SUBAPPLICATION Uebung_221 (* Standard IEC 61131-3 FB_CTUD_DINT (Vor-/Rückwärtszähler, DINT) mit Terminal-Ausgabe *)
  (* Standard: 61131-3; Description: Copyright (c) 2026 Meisterschulen am Ostbahnhof This program and the accompanying materials are made available under the terms of the Eclipse Public License 2.0 which is available at https://www.eclipse.org/legal/epl-2.0/ SPDX-License-Identifier: EPL-2.0 *)
  (* Version 1.1, 2026-04-21, Franz Höpfinger, Meisterschulen am Ostbahnhof, Added terminal output for counter value *)
  (* Version 1.0, 2026-04-20, Franz Höpfinger, Meisterschulen am Ostbahnhof, initial API and implementation (IEC 61131-3 version) *)
  PACKAGE Uebungen;
  IMPORT Uebungen::const::UT::DefaultPool::OutputNumber_N1;
  IMPORT logiBUS::io::DI::logiBUS_DI::Input_I1;
  IMPORT logiBUS::io::DI::logiBUS_DI::Input_I2;
  IMPORT logiBUS::io::DI::logiBUS_DI::Input_I3;
  IMPORT logiBUS::io::DI::logiBUS_DI::Input_I4;
  IMPORT logiBUS::io::DQ::logiBUS_DO::Output_Q1;
  IMPORT logiBUS::io::DQ::logiBUS_DO::Output_Q2;
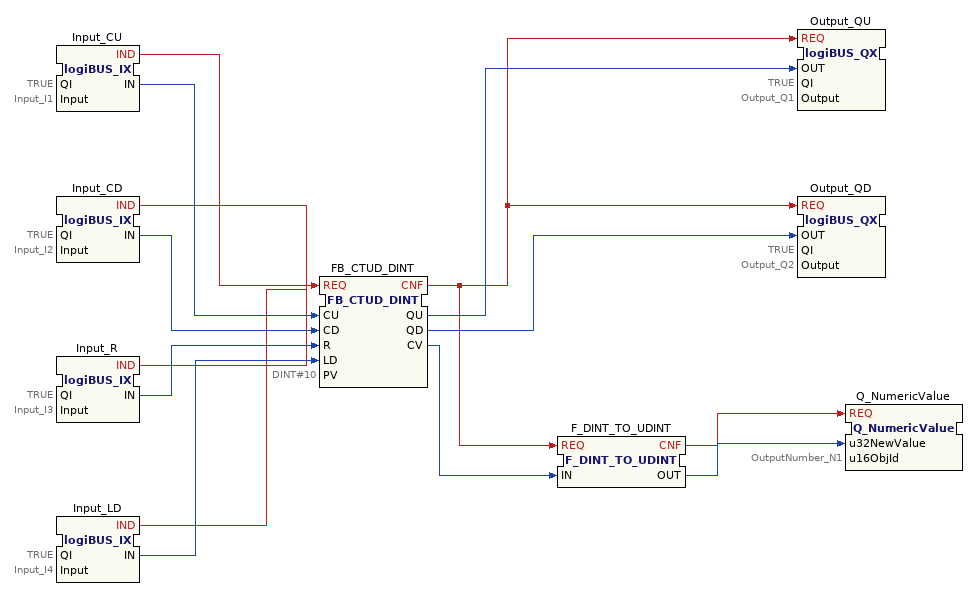
  (* F_DINT_TO_UDINT ist großer Quatsch ... keine Negativen Zahlen möglich *)
  FBS
    FB_CTUD_DINT : iec61131::counters::FB_CTUD_DINT(PV := DINT#10);
    Input_CU : logiBUS::io::DI::logiBUS_IX(QI := TRUE, Input := Input_I1);
    Input_CD : logiBUS::io::DI::logiBUS_IX(QI := TRUE, Input := Input_I2);
    Input_R : logiBUS::io::DI::logiBUS_IX(QI := TRUE, Input := Input_I3);
    Input_LD : logiBUS::io::DI::logiBUS_IX(QI := TRUE, Input := Input_I4);
    Output_QU : logiBUS::io::DQ::logiBUS_QX(QI := TRUE, Output := Output_Q1);
    Output_QD : logiBUS::io::DQ::logiBUS_QX(QI := TRUE, Output := Output_Q2);
    Q_NumericValue : isobus::UT::Q::Q_NumericValue(u16ObjId := OutputNumber_N1);
    F_DINT_TO_UDINT : iec61131::conversion::F_DINT_TO_UDINT;
  END_FBS
  EVENT_CONNECTIONS
    Input_CU.IND TO FB_CTUD_DINT.REQ;
    Input_CD.IND TO FB_CTUD_DINT.REQ;
    Input_R.IND TO FB_CTUD_DINT.REQ;
    Input_LD.IND TO FB_CTUD_DINT.REQ;
    FB_CTUD_DINT.CNF TO Output_QU.REQ;
    FB_CTUD_DINT.CNF TO Output_QD.REQ;
    FB_CTUD_DINT.CNF TO F_DINT_TO_UDINT.REQ;
    F_DINT_TO_UDINT.CNF TO Q_NumericValue.REQ;
  END_CONNECTIONS
  DATA_CONNECTIONS
    Input_CU.IN TO FB_CTUD_DINT.CU;
    Input_CD.IN TO FB_CTUD_DINT.CD;
    Input_R.IN TO FB_CTUD_DINT.R;
    Input_LD.IN TO FB_CTUD_DINT.LD;
    FB_CTUD_DINT.QU TO Output_QU.OUT;
    FB_CTUD_DINT.QD TO Output_QD.OUT;
    FB_CTUD_DINT.CV TO F_DINT_TO_UDINT.IN;
    F_DINT_TO_UDINT.OUT TO Q_NumericValue.u32NewValue;
  END_CONNECTIONS
END_SUBAPPLICATION
